Staubli VAL3: gestureFist.pgx

program gestureFist()
begin
  //close(tClaw)



  if (bClawClosed==false)
  close(tClaw)
  putln("Fist Closed")
  bClawClosed=true
  elseIf (bClawClosed==true)
  open(tClaw)
  putln("Fist Opened")
  bClawClosed=false
  endIf
end
